# EPICS autosave request: apps/XY560App/Db/XY560_chN_settings.req
# XY560_chN_settings.req - XY560 32-Channel Analog Input Module
$(P)$(R)_$(C)_$(N).DESC
$(P)$(R)_$(C)_$(N).LINR
$(P)$(R)_$(C)_$(N).EGUF
$(P)$(R)_$(C)_$(N).EGUL
$(P)$(R)_$(C)_$(N).EGU
$(P)$(R)_$(C)_$(N).PREC
$(P)$(R)_$(C)_$(N).HOPR
$(P)$(R)_$(C)_$(N).LOPR
# alarms
$(P)$(R)_$(C)_$(N).HIHI
$(P)$(R)_$(C)_$(N).HIGH
$(P)$(R)_$(C)_$(N).LOW
$(P)$(R)_$(C)_$(N).LOLO
$(P)$(R)_$(C)_$(N).HHSV
$(P)$(R)_$(C)_$(N).HSV
$(P)$(R)_$(C)_$(N).LSV
$(P)$(R)_$(C)_$(N).LLSV
